FUNCTION_BLOCK AE_TO_AE2 (* Composite FB for convert unidirectional AE to bidirectional AE2 *)
  (* Standard: 61499-2; Function: AE_IN publishes its event onto the outgoing (EO1) side of AE2_BIDIR. Whatever AE2_BIDIR receives on its incoming (EI1) side is forwarded out again as a plain unidirectional event via AE_OUT.; Description: Copyright (c) 2026 HR Agrartechnik GmbH This program and the accompanying materials are made available under the terms of the Eclipse Public License 2.0 which is available at https://www.eclipse.org/legal/epl-2.0/ SPDX-License-Identifier: EPL-2.0 *)
  (* Version 1.0, 2026-08-31, Franz Höpfinger, HR Agrartechnik GmbH, Initial Version *)
  PACKAGE adapter::conversion::bidirectional;
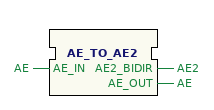
  SOCKETS
    AE_IN : adapter::types::unidirectional::AE; (* Adapter Input: unidirectional source *)
  END_SOCKETS
  PLUGS
    AE2_BIDIR : adapter::types::bidirectional::AE2; (* Adapter Output: bidirectional tap, outgoing side driven by AE_IN, incoming side forwarded to AE_OUT *)
    AE_OUT : adapter::types::unidirectional::AE; (* Adapter Output: mirrors AE2_BIDIR's incoming (request) side *)
  END_PLUGS
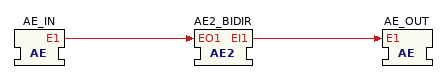
  EVENT_CONNECTIONS
    AE_IN.E1 TO AE2_BIDIR.EO1;
    AE2_BIDIR.EI1 TO AE_OUT.E1;
  END_CONNECTIONS
END_FUNCTION_BLOCK
